{attribute 'qualified_only'}
VAR_GLOBAL
END_VAR

(* stored: Version 1.1.0.1, ProductVersion 3.1.4024.16
   GVL Nums: Id {8deb4d67-9560-41b5-b7b6-4fa285b12493} *)
